DATA_BLOCK DB 3
AUTHOR : sra
FAMILY : AZO
VERSION : 0.0
  STRUCT
   OB1_Info : STRUCT
    OB1_DATE_TIME : DATE_AND_TIME ;	//Date and time OB1 started
    OB1_PREV_CYCLE : INT ;	//Cycle time of previous OB1 scan (milliseconds)
    OB1_MIN_CYCLE : INT ;	//Minimum cycle time of OB1 (milliseconds)
    OB1_MAX_CYCLE : INT ;	//Maximum cycle time of OB1 (milliseconds)
    reserve : ARRAY  [0 .. 14 ] OF BYTE ;
   END_STRUCT ;
   Fehler_OB_Info : STRUCT
    Zeitfehler_OB80 : BOOL ;	//Zeitfehler OB 80
    Stromversorgung_OB81 : BOOL ;	//Stromversorgungsfehler OB 81
    Diagnose_Alarm_OB82 : BOOL ;	//Diagnose-Alarm OB82
    Ziehen_Stecken_OB83 : BOOL ;	//Ziehen/Stecken-Alarm OB83
    CPU_Hardware_OB84 : BOOL ;	//CPU-Hardwarefehler OB84
    Programmablauf_OB85 : BOOL ;	//Programmablauffehler OB85
    Baugr_tr_ausfall_OB86 : BOOL ;	//Baugruppenträgerausfall OB86
    Kommunikation_OB87 : BOOL ;	//Kommunikationsfehler OB87
    Programmierfehler_OB121 : BOOL ;	//Programmierfehler OB121
    Periphzugriff_OB122 : BOOL ;	//Peripheriezugriffsfehler OB 122
    Bearbeitungsabbruch_OB88 : BOOL ;	//Bearbeitungsabbruch eines Bausteins OB88
    Battery_fault : BOOL ;	//Battery fault with SFC51
    reserve_word : WORD ;
    OB_80_Fault_ID : BYTE ;	//Fehlercode OB 80
    OB_81_Fault_ID : BYTE ;	//Fehlercode OB 81
    OB_82_Fault_ID : BYTE ;	//Fehlercode OB 82
    OB_83_Fault_ID : BYTE ;	//Fehlercode OB 83
    OB_84_Fault_ID : BYTE ;	//Fehlercode OB 84
    OB_85_Fault_ID : BYTE ;	//Fehlercode OB 85
    OB_86_Fault_ID : BYTE ;	//Fehlercode OB 86
    OB_87_Fault_ID : BYTE ;	//Fehlercode OB 87
    OB_121_Fault_ID : BYTE ;	//Fehlercode OB 121
    OB_122_Fault_ID : BYTE ;	//Fehlercode OB 122
    OB_88_Fault_ID : BYTE ;	//Fehlercode OB 122
    reserve : ARRAY  [16 .. 29 ] OF BYTE ;
   END_STRUCT ;
   RDSYSST : STRUCT
    BUSY : BOOL ;
    RETVAL : INT ;
    SLZ_HEADER : STRUCT
     LENTHDR : WORD ;
     N_DR : WORD ;
    END_STRUCT ;
    DR : STRUCT
     Data_1 : BYTE ;
     Data_2 : BYTE ;
     Data_3 : BYTE ;
     Data_4 : BYTE ;
     Data_5 : BYTE ;
     Data_6 : BYTE ;
     Data_7 : BYTE ;
     Data_8 : BYTE ;
     Data_9 : BYTE ;
     Data_10 : BYTE ;
     Data_11 : BYTE ;
     Data_12 : BYTE ;
     Data_13 : BYTE ;
     Data_14 : BYTE ;
     Data_15 : BYTE ;
     Data_16 : BYTE ;
     Data_17 : BYTE ;
     Data_18 : BYTE ;
     Data_19 : BYTE ;
     Data_20 : BYTE ;
    END_STRUCT ;
   END_STRUCT ;
  END_STRUCT ;	
BEGIN
END_DATA_BLOCK

DATA_BLOCK DB 4
VERSION : 0.1
  STRUCT
   Motordaten1 : STRUCT 	//Anzahl der Motordaten abhängig von der Anzahl der verschied. benutzten Motoren
    Nennleistungsfaktor : REAL  := 8.000000e-001;	//Motornennleistungsfaktor cos phi
    Nennfrequenz : REAL  := 5.100000e+001;	//Motornennfrequenz in Einheit Hz
    Nenndrehzahl : REAL  := 1.400000e+003;	//Motornenndrehzal in U/min
    Nennstrom : REAL  := 6.100000e+000;	//Motornennstrom in A
    Nennspannung : REAL  := 2.310000e+002;	//Motornennspannung in V
    Nennleistung : REAL  := 1.400000e+000;	//Motornennleistung kW
    reserve : ARRAY  [24 .. 29 ] OF //Reserve für weitere Motordaten
    BYTE ;
   END_STRUCT ;
   Motordaten2 : STRUCT
    Nennleistungsfaktor : REAL  := 7.000000e-001;
    Nennfrequenz : REAL  := 1.000000e+002;
    Nenndrehzahl : REAL  := 2.000000e+002;
    Nennstrom : REAL  := 2.000000e+000;
    Nennspannung : REAL  := 3.800000e+002;
    Nennleistung : REAL  := 1.000000e+003;
    reserve : ARRAY  [24 .. 29 ] OF BYTE ;
   END_STRUCT ;
   Motordaten3 : STRUCT
    Nennleistungsfaktor : REAL  := 7.000000e-001;
    Nennfrequenz : REAL  := 1.000000e+002;
    Nenndrehzahl : REAL  := 2.000000e+002;
    Nennstrom : REAL  := 5.000000e+000;
    Nennspannung : REAL  := 3.800000e+002;
    Nennleistung : REAL  := 1.000000e+003;
    reserve : ARRAY  [24 .. 29 ] OF BYTE ;
   END_STRUCT ;
   Motordaten4 : STRUCT
    Nennleistungsfaktor : REAL  := 7.000000e-001;
    Nennfrequenz : REAL  := 1.000000e+002;
    Nenndrehzahl : REAL  := 2.000000e+002;
    Nennstrom : REAL  := 5.000000e+000;
    Nennspannung : REAL  := 3.800000e+002;
    Nennleistung : REAL  := 1.000000e+003;
    reserve : ARRAY  [24 .. 29 ] OF BYTE ;
   END_STRUCT ;
   Motordaten5 : STRUCT
    Nennleistungsfaktor : REAL  := 7.000000e-001;
    Nennfrequenz : REAL  := 1.000000e+002;
    Nenndrehzahl : REAL  := 2.000000e+002;
    Nennstrom : REAL  := 5.000000e+000;
    Nennspannung : REAL  := 3.800000e+002;
    Nennleistung : REAL  := 1.000000e+003;
    reserve : ARRAY  [24 .. 29 ] OF BYTE ;
   END_STRUCT ;
   Motordaten6 : STRUCT
    Nennleistungsfaktor : REAL  := 7.000000e-001;
    Nennfrequenz : REAL  := 1.000000e+002;
    Nenndrehzahl : REAL  := 2.000000e+002;
    Nennstrom : REAL  := 5.000000e+000;
    Nennspannung : REAL  := 3.800000e+002;
    Nennleistung : REAL  := 1.000000e+003;
    reserve : ARRAY  [24 .. 29 ] OF BYTE ;
   END_STRUCT ;
   Motordaten7 : STRUCT
    Nennleistungsfaktor : REAL  := 7.000000e-001;
    Nennfrequenz : REAL  := 1.000000e+002;
    Nenndrehzahl : REAL  := 2.000000e+002;
    Nennstrom : REAL  := 5.000000e+000;
    Nennspannung : REAL  := 3.800000e+002;
    Nennleistung : REAL  := 1.000000e+003;
    reserve : ARRAY  [24 .. 29 ] OF BYTE ;
   END_STRUCT ;
   Motordaten8 : STRUCT
    Nennleistungsfaktor : REAL  := 7.000000e-001;
    Nennfrequenz : REAL  := 1.000000e+002;
    Nenndrehzahl : REAL  := 2.000000e+002;
    Nennstrom : REAL  := 5.000000e+000;
    Nennspannung : REAL  := 3.800000e+002;
    Nennleistung : REAL  := 1.000000e+003;
    reserve : ARRAY  [24 .. 29 ] OF BYTE ;
   END_STRUCT ;
   Motordaten9 : STRUCT
    Nennleistungsfaktor : REAL  := 7.000000e-001;
    Nennfrequenz : REAL  := 1.000000e+002;
    Nenndrehzahl : REAL  := 2.000000e+002;
    Nennstrom : REAL  := 5.000000e+000;
    Nennspannung : REAL  := 3.800000e+002;
    Nennleistung : REAL  := 1.000000e+003;
    reserve : ARRAY  [24 .. 29 ] OF BYTE ;
   END_STRUCT ;
   Motordaten10 : STRUCT
    Nennleistungsfaktor : REAL  := 7.000000e-001;
    Nennfrequenz : REAL  := 1.000000e+002;
    Nenndrehzahl : REAL  := 2.000000e+002;
    Nennstrom : REAL  := 5.000000e+000;
    Nennspannung : REAL  := 3.800000e+002;
    Nennleistung : REAL  := 1.000000e+003;
    reserve : ARRAY  [24 .. 29 ] OF BYTE ;
   END_STRUCT ;
  END_STRUCT ;	
BEGIN
   Motordaten1.Nennleistungsfaktor := 8.000000e-01;
   Motordaten1.Nennfrequenz := 5.100000e+01;
   Motordaten1.Nenndrehzahl := 1.400000e+03;
   Motordaten1.Nennstrom := 6.100000e+00;
   Motordaten1.Nennspannung := 2.310000e+02;
   Motordaten1.Nennleistung := 1.400000e+00;
   Motordaten2.Nennleistungsfaktor := 7.000000e-01;
   Motordaten2.Nennfrequenz := 1.000000e+02;
   Motordaten2.Nenndrehzahl := 2.000000e+02;
   Motordaten2.Nennstrom := 5.000000e+00;
   Motordaten2.Nennspannung := 3.800000e+02;
   Motordaten2.Nennleistung := 1.000000e+03;
   Motordaten3.Nennleistungsfaktor := 7.000000e-01;
   Motordaten3.Nennfrequenz := 1.000000e+02;
   Motordaten3.Nenndrehzahl := 2.000000e+02;
   Motordaten3.Nennstrom := 5.000000e+00;
   Motordaten3.Nennspannung := 3.800000e+02;
   Motordaten3.Nennleistung := 1.000000e+03;
   Motordaten4.Nennleistungsfaktor := 7.000000e-01;
   Motordaten4.Nennfrequenz := 1.000000e+02;
   Motordaten4.Nenndrehzahl := 2.000000e+02;
   Motordaten4.Nennstrom := 5.000000e+00;
   Motordaten4.Nennspannung := 3.800000e+02;
   Motordaten4.Nennleistung := 1.000000e+03;
   Motordaten5.Nennleistungsfaktor := 7.000000e-01;
   Motordaten5.Nennfrequenz := 1.000000e+02;
   Motordaten5.Nenndrehzahl := 2.000000e+02;
   Motordaten5.Nennstrom := 5.000000e+00;
   Motordaten5.Nennspannung := 3.800000e+02;
   Motordaten5.Nennleistung := 1.000000e+03;
   Motordaten6.Nennleistungsfaktor := 7.000000e-01;
   Motordaten6.Nennfrequenz := 1.000000e+02;
   Motordaten6.Nenndrehzahl := 2.000000e+02;
   Motordaten6.Nennstrom := 5.000000e+00;
   Motordaten6.Nennspannung := 3.800000e+02;
   Motordaten6.Nennleistung := 1.000000e+03;
   Motordaten7.Nennleistungsfaktor := 7.000000e-01;
   Motordaten7.Nennfrequenz := 1.000000e+02;
   Motordaten7.Nenndrehzahl := 2.000000e+02;
   Motordaten7.Nennstrom := 5.000000e+00;
   Motordaten7.Nennspannung := 3.800000e+02;
   Motordaten7.Nennleistung := 1.000000e+03;
   Motordaten8.Nennleistungsfaktor := 7.000000e-01;
   Motordaten8.Nennfrequenz := 1.000000e+02;
   Motordaten8.Nenndrehzahl := 2.000000e+02;
   Motordaten8.Nennstrom := 5.000000e+00;
   Motordaten8.Nennspannung := 3.800000e+02;
   Motordaten8.Nennleistung := 1.000000e+03;
   Motordaten9.Nennleistungsfaktor := 7.000000e-01;
   Motordaten9.Nennfrequenz := 1.000000e+02;
   Motordaten9.Nenndrehzahl := 2.000000e+02;
   Motordaten9.Nennstrom := 5.000000e+00;
   Motordaten9.Nennspannung := 3.800000e+02;
   Motordaten9.Nennleistung := 1.000000e+03;
   Motordaten10.Nennleistungsfaktor := 7.000000e-01;
   Motordaten10.Nennfrequenz := 1.000000e+02;
   Motordaten10.Nenndrehzahl := 2.000000e+02;
   Motordaten10.Nennstrom := 5.000000e+00;
   Motordaten10.Nennspannung := 3.800000e+02;
   Motordaten10.Nennleistung := 1.000000e+03;
END_DATA_BLOCK

DATA_BLOCK DB 30
AUTHOR : sra
FAMILY : hsh
VERSION : 0.0
FB 30
BEGIN
END_DATA_BLOCK

DATA_BLOCK DB 32
AUTHOR : sra
FAMILY : SCADA
VERSION : 0.0
FB 32
BEGIN
END_DATA_BLOCK

DATA_BLOCK DB 33
AUTHOR : sra
FAMILY : SCADA
VERSION : 0.0
FB 33
BEGIN
END_DATA_BLOCK

DATA_BLOCK DB 34
AUTHOR : sra
FAMILY : AZO
VERSION : 0.0
FB 34
BEGIN
END_DATA_BLOCK

DATA_BLOCK DB 35
VERSION : 0.1
  STRUCT
   Quittierung : ARRAY  [0 .. 1023, 0 .. 7 ] OF BOOL  := FALSE;
   Quittierung_Spiegelungen : ARRAY  [0 .. 1023, 0 .. 7 ] OF BOOL  := FALSE;
  END_STRUCT ;	
BEGIN
END_DATA_BLOCK

DATA_BLOCK DB 92
VERSION : 0.0
FB 92
BEGIN
END_DATA_BLOCK

DATA_BLOCK DB 1000
AUTHOR : ilia
VERSION : 0.0
FB 1000
BEGIN
END_DATA_BLOCK

DATA_BLOCK DB 1001
AUTHOR : ilia
VERSION : 0.1
FB 1001
BEGIN
END_DATA_BLOCK

DATA_BLOCK DB 1011
AUTHOR : ilia
VERSION : 0.1
FB 1011
BEGIN
END_DATA_BLOCK

DATA_BLOCK DB 1051
AUTHOR : ilia
VERSION : 0.1
FB 1051
BEGIN
END_DATA_BLOCK

DATA_BLOCK DB 1111
VERSION : 0.1
  STRUCT
   RECIPE1 : STRUCT 	//Recipe
    RecipeName : STRING  [18 ] := 'RECIPE1';	//Recipe Name
    SpeedRinne : INT  := 30;	//Speed of Rinne
    SpeedRotaryFeeder : INT  := 30;	//Speed of RF
    SpeedVacuumPump : INT  := 35;	//Speed of VP1
    NumberOfPumps : INT  := 1;
    reserve1 : INT ;
    reserve2 : INT ;
    reserve3 : ARRAY  [1 .. 8 ] OF BYTE  := B#16#0;
   END_STRUCT ;
   RECIPE2 : STRUCT 	//Recipe
    RecipeName : STRING  [18 ] := 'RECIPE2';	//Recipe Name
    SpeedRinne : INT  := 30;	//Speed of Rinne
    SpeedRotaryFeeder : INT  := 30;	//Speed of RF
    SpeedVacuumPump : INT  := 35;	//Speed of VP1
    NumberOfPumps : INT  := 1;
    reserve1 : INT ;
    reserve2 : INT ;
    reserve3 : ARRAY  [1 .. 8 ] OF BYTE  := B#16#0;
   END_STRUCT ;
   RECIPE3 : STRUCT 	//Recipe
    RecipeName : STRING  [18 ] := 'RECIPE3';	//Recipe Name
    SpeedRinne : INT  := 30;	//Speed of Rinne
    SpeedRotaryFeeder : INT  := 30;	//Speed of RF
    SpeedVacuumPump : INT  := 35;	//Speed of VP1
    NumberOfPumps : INT  := 1;
    reserve1 : INT ;
    reserve2 : INT ;
    reserve3 : ARRAY  [1 .. 8 ] OF BYTE  := B#16#0;
   END_STRUCT ;
   RECIPE4 : STRUCT 	//Recipe
    RecipeName : STRING  [18 ] := 'RECIPE4';	//Recipe Name
    SpeedRinne : INT  := 30;	//Speed of Rinne
    SpeedRotaryFeeder : INT  := 30;	//Speed of RF
    SpeedVacuumPump : INT  := 35;	//Speed of VP1
    NumberOfPumps : INT  := 1;
    reserve1 : INT ;
    reserve2 : INT ;
    reserve3 : ARRAY  [1 .. 8 ] OF BYTE  := B#16#0;
   END_STRUCT ;
   RECIPE5 : STRUCT 	//Recipe
    RecipeName : STRING  [18 ] := 'RECIPE5';	//Recipe Name
    SpeedRinne : INT  := 30;	//Speed of Rinne
    SpeedRotaryFeeder : INT  := 30;	//Speed of RF
    SpeedVacuumPump : INT  := 35;	//Speed of VP1
    NumberOfPumps : INT  := 1;
    reserve1 : INT ;
    reserve2 : INT ;
    reserve3 : ARRAY  [1 .. 8 ] OF BYTE  := B#16#0;
   END_STRUCT ;
   RECIPE6 : STRUCT 	//Recipe
    RecipeName : STRING  [18 ] := 'RECIPE6';	//Recipe Name
    SpeedRinne : INT  := 30;	//Speed of Rinne
    SpeedRotaryFeeder : INT  := 30;	//Speed of RF
    SpeedVacuumPump : INT  := 35;	//Speed of VP1
    NumberOfPumps : INT  := 1;
    reserve1 : INT ;
    reserve2 : INT ;
    reserve3 : ARRAY  [1 .. 8 ] OF BYTE  := B#16#0;
   END_STRUCT ;
   RECIPE7 : STRUCT 	//Recipe
    RecipeName : STRING  [18 ] := 'RECIPE7';	//Recipe Name
    SpeedRinne : INT  := 30;	//Speed of Rinne
    SpeedRotaryFeeder : INT  := 30;	//Speed of RF
    SpeedVacuumPump : INT  := 35;	//Speed of VP1
    NumberOfPumps : INT  := 1;
    reserve1 : INT ;
    reserve2 : INT ;
    reserve3 : ARRAY  [1 .. 8 ] OF BYTE  := B#16#0;
   END_STRUCT ;
   RECIPE8 : STRUCT 	//Recipe
    RecipeName : STRING  [18 ] := 'RECIPE8';	//Recipe Name
    SpeedRinne : INT  := 30;	//Speed of Rinne
    SpeedRotaryFeeder : INT  := 30;	//Speed of RF
    SpeedVacuumPump : INT  := 35;	//Speed of VP1
    NumberOfPumps : INT  := 1;
    reserve1 : INT ;
    reserve2 : INT ;
    reserve3 : ARRAY  [1 .. 8 ] OF BYTE  := B#16#0;
   END_STRUCT ;
   RECIPE9 : STRUCT 	//Recipe
    RecipeName1 : STRING  [18 ] := 'RECIPE9';	//Recipe Name
    SpeedRinne : INT  := 30;	//Speed of Rinne
    SpeedRotaryFeeder : INT  := 30;	//Speed of RF
    SpeedVacuumPump : INT  := 35;	//Speed of VP1
    NumberOfPumps : INT  := 1;
    reserve1 : INT ;
    reserve2 : INT ;
    reserve3 : ARRAY  [1 .. 8 ] OF BYTE  := B#16#0;
   END_STRUCT ;
   RECIPE10 : STRUCT 	//Recipe
    RecipeName : STRING  [18 ] := 'RECIPE10';	//Recipe Name
    SpeedRinne : INT  := 30;	//Speed of Rinne
    SpeedRotaryFeeder : INT  := 30;	//Speed of RF
    SpeedVacuumPump : INT  := 35;	//Speed of VP1
    NumberOfPumps : INT  := 1;
    reserve1 : INT ;
    reserve2 : INT ;
    reserve3 : ARRAY  [1 .. 8 ] OF BYTE  := B#16#0;
   END_STRUCT ;
  END_STRUCT ;	
BEGIN
   RECIPE1.RecipeName := 'RECIPE1';
   RECIPE1.SpeedRinne := 30;
   RECIPE1.SpeedRotaryFeeder := 30;
   RECIPE1.SpeedVacuumPump := 35;
   RECIPE1.NumberOfPumps := 1;
   RECIPE2.RecipeName := 'RECIPE2';
   RECIPE2.SpeedRinne := 30;
   RECIPE2.SpeedRotaryFeeder := 30;
   RECIPE2.SpeedVacuumPump := 35;
   RECIPE2.NumberOfPumps := 1;
   RECIPE3.RecipeName := 'RECIPE3';
   RECIPE3.SpeedRinne := 30;
   RECIPE3.SpeedRotaryFeeder := 30;
   RECIPE3.SpeedVacuumPump := 35;
   RECIPE3.NumberOfPumps := 1;
   RECIPE4.RecipeName := 'RECIPE4';
   RECIPE4.SpeedRinne := 30;
   RECIPE4.SpeedRotaryFeeder := 30;
   RECIPE4.SpeedVacuumPump := 35;
   RECIPE4.NumberOfPumps := 1;
   RECIPE5.RecipeName := 'RECIPE5';
   RECIPE5.SpeedRinne := 30;
   RECIPE5.SpeedRotaryFeeder := 30;
   RECIPE5.SpeedVacuumPump := 35;
   RECIPE5.NumberOfPumps := 1;
   RECIPE6.RecipeName := 'RECIPE6';
   RECIPE6.SpeedRinne := 30;
   RECIPE6.SpeedRotaryFeeder := 30;
   RECIPE6.SpeedVacuumPump := 35;
   RECIPE6.NumberOfPumps := 1;
   RECIPE7.RecipeName := 'RECIPE7';
   RECIPE7.SpeedRinne := 30;
   RECIPE7.SpeedRotaryFeeder := 30;
   RECIPE7.SpeedVacuumPump := 35;
   RECIPE7.NumberOfPumps := 1;
   RECIPE8.RecipeName := 'RECIPE8';
   RECIPE8.SpeedRinne := 30;
   RECIPE8.SpeedRotaryFeeder := 30;
   RECIPE8.SpeedVacuumPump := 35;
   RECIPE8.NumberOfPumps := 1;
   RECIPE9.RecipeName1 := 'RECIPE9';
   RECIPE9.SpeedRinne := 30;
   RECIPE9.SpeedRotaryFeeder := 30;
   RECIPE9.SpeedVacuumPump := 35;
   RECIPE9.NumberOfPumps := 1;
   RECIPE10.RecipeName := 'RECIPE10';
   RECIPE10.SpeedRinne := 30;
   RECIPE10.SpeedRotaryFeeder := 30;
   RECIPE10.SpeedVacuumPump := 35;
   RECIPE10.NumberOfPumps := 1;
END_DATA_BLOCK

DATA_BLOCK DB 2222
VERSION : 0.1
  STRUCT
   Recipe : STRUCT 	//Temporary placeholder variable
    Speed_1 : INT  := 1;
    Speed_2 : INT  := 2;
    Number : INT ;
   END_STRUCT ;
  END_STRUCT ;	
BEGIN
   Recipe.Speed_1 := 1;
   Recipe.Speed_2 := 2;
END_DATA_BLOCK

DATA_BLOCK DB 4900
AUTHOR : ilia
VERSION : 0.0
FB 4900
BEGIN
END_DATA_BLOCK

DATA_BLOCK DB 10001
VERSION : 0.0
FB 4901
BEGIN
END_DATA_BLOCK

DATA_BLOCK DB 10002
VERSION : 0.0
FB 4901
BEGIN
END_DATA_BLOCK

ORGANIZATION_BLOCK OB 1
TITLE = zyklischer Programmablauf
//Erstellung:
//Datum        Bearbeiter                                                 Version
//--------------------------------------------------------------------------------
//01.08.18     Ilia Bedniakov                                             01.00.00
//
//Änderungen:
//Nr. Datum    Bearb Beschreibung                                   Marke Version
//--------------------------------------------------------------------------------
//01  
//
VERSION : 0.1
VAR_TEMP
  OB1_EV_CLASS : BYTE ;	//Bits 0-3 = 1 (Coming event), Bits 4-7 = 1 (Event class 1)
  OB1_SCAN_1 : BYTE ;	//1 (Cold restart scan 1 of OB 1), 3 (Scan 2-n of OB 1)
  OB1_PRIORITY : BYTE ;	//1 (Priority of 1 is lowest)
  OB1_OB_NUMBR : BYTE ;	//1 (Organization block 1, OB1)
  OB1_RESERVED_1 : BYTE ;	//Reserved for system
  OB1_RESERVED_2 : BYTE ;	//Reserved for system
  OB1_PREV_CYCLE : INT ;	//Cycle time of previous OB1 scan (milliseconds)
  OB1_MIN_CYCLE : INT ;	//Minimum cycle time of OB1 (milliseconds)
  OB1_MAX_CYCLE : INT ;	//Maximum cycle time of OB1 (milliseconds)
  OB1_DATE_TIME : DATE_AND_TIME ;	//Date and time OB1 started
  DUMMY_INT : INT ;
  dummybool : BOOL ;
END_VAR
BEGIN
NETWORK
TITLE = Simulation
//      CLR   
      SET;
      =     M 0.5;
      A     M 0.5;
      JCN   NS;	// No simulation
      CALL  FB 2 , DB 2;
NS:   NOP   0;
NETWORK
TITLE = Datum, Uhrzeit und Zykluszeiten in DB3 kopieren
      CALL  SFC 20 (
           SRCBLK                   := #OB1_DATE_TIME,
           RET_VAL                  := #DUMMY_INT,
           DSTBLK                   := P#DB3.DBX 0.0 BYTE 8);
      L     #OB1_PREV_CYCLE;
      T     DB3.DBW 8;
      L     #OB1_MIN_CYCLE;
      T     DB3.DBW 10;
      L     #OB1_MAX_CYCLE;
      T     DB3.DBW 12;
NETWORK
TITLE = Standardsignale
      CALL  FC 13 (
           in_E_Sicherung_OK        := I 5.7,
           in_Basistakt_Timer       := M 4.1,
           in_Zeit_Basistakt_100ms  := 2,
           o_Lampe_Stoer_Sicherung  := #dummybool,
           o_Stoerung_Sicherung     := #dummybool);
NETWORK
TITLE = Daten von/an HMI
      CALL  FB 30 , DB 30;
      CALL  FB 32 , DB 32;
      CALL  FB 33 , DB 33;
NETWORK
TITLE = Stoerungen Auswertung
      CALL  FB 34 , DB 34;
NETWORK
TITLE = Anwenderprogramm
      CALL  FB 1000 , DB 1000;
NETWORK
TITLE = Neustart oder Wiederanlauf SPS rücksetzen
//letztes Netzwerk
      SET;
      R     M 1.3;
      R     M 1.4;
END_ORGANIZATION_BLOCK

ORGANIZATION_BLOCK OB 80
TITLE = Zeitfehler
//Erstellung:
//Datum        Bearbeiter                                                 Version
//--------------------------------------------------------------------------------
//03.06.98     Rainer Schaffert (sra)                                     01.00.00
//
//Änderungen:
//Nr. Datum    Bearb Beschreibung                                   Marke Version
//--------------------------------------------------------------------------------
//01  
//
//________________________________________________________________________________
//OB wird bei Zeitfehler bearbeitet
//
AUTHOR : sra
FAMILY : error_OB
NAME : time_err
VERSION : 0.1
VAR_TEMP
  OB80_EV_CLASS : BYTE ;	//16#35, Event class 3, Entering event state, Internal fault event
  OB80_FLT_ID : BYTE ;	//16#XX, Fault identifcation code
  OB80_PRIORITY : BYTE ;	//26 (Priority of 1 is lowest)
  OB80_OB_NUMBR : BYTE ;	//80 (Organization block 80, OB80)
  OB80_RESERVED_1 : BYTE ;	//Reserved for system
  OB80_RESERVED_2 : BYTE ;	//Reserved for system
  OB80_ERROR_INFO : WORD ;	//Error information on event
  OB80_ERR_EV_CLASS : BYTE ;	//Class of event causing error
  OB80_ERR_EV_NUM : BYTE ;	//Number of event causing error
  OB80_OB_PRIORITY : BYTE ;	//Priority of OB causing error
  OB80_OB_NUM : BYTE ;	//Number of OB causing error
  OB80_DATE_TIME : DATE_AND_TIME ;	//Date and time OB80 started
END_VAR
BEGIN
NETWORK
TITLE = Fehlermeldung erzeugen
//Fehlermeldung erzeugen
//
//Fehlercode B#16#01 : Zykluszeit überschritten
//                     OB80_ERROR_INFO: Laufzeit des letzten Zyklus
//           
//           B#16#02 : Der angeforderte OB ist noch in Bearbeitung
//
//           B#16#07 : Überlauf des OB-Anforderungspuffers für die aktuelle 
//                     Prioritätsklasse
//
//           B#16#05 : abgelaufener Urzeitalarm durch Urzeitsprung
//
//           B#16#06 : abgelaufener Urzeitalarm bei Wiedereintritt 
//
      L     #OB80_FLT_ID;
      L     B#16#0;
      <>I;
      =     DB3.DBX 30.0;
      L     #OB80_FLT_ID;
      T     DB3.DBB 34;
END_ORGANIZATION_BLOCK

ORGANIZATION_BLOCK OB 82
TITLE = Diagnose-Alarm
//Erstellung:
//Datum        Bearbeiter                                                 Version
//--------------------------------------------------------------------------------
//03.06.98     Rainer Schaffert (sra)                                     01.00.00
//
//Änderungen:
//Nr. Datum    Bearb Beschreibung                                   Marke Version
//--------------------------------------------------------------------------------
//01  
//
//________________________________________________________________________________
//OB wird bei Diagnose-Alarm bearbeitet
//
AUTHOR : sra
FAMILY : error_OB
NAME : diagn_OB
VERSION : 0.1
VAR_TEMP
  OB82_EV_CLASS : BYTE ;	//16#39, Event class 3, Entering event state, Internal fault event
  OB82_FLT_ID : BYTE ;	//16#XX, Fault identifcation code
  OB82_PRIORITY : BYTE ;	//26/28 (Priority of 1 is lowest)
  OB82_OB_NUMBR : BYTE ;	//82 (Organization block 82, OB82)
  OB82_RESERVED_1 : BYTE ;	//Reserved for system
  OB82_IO_FLAG : BYTE ;	//Input (01010100), Output (01010101)
  OB82_MDL_ADDR : INT ;	//Base address of module with fault
  OB82_MDL_DEFECT : BOOL ;	//Module defective
  OB82_INT_FAULT : BOOL ;	//Internal fault
  OB82_EXT_FAULT : BOOL ;	//External fault
  OB82_PNT_INFO : BOOL ;	//Point information
  OB82_EXT_VOLTAGE : BOOL ;	//External voltage low
  OB82_FLD_CONNCTR : BOOL ;	//Field wiring connector missing
  OB82_NO_CONFIG : BOOL ;	//Module has no configuration data
  OB82_CONFIG_ERR : BOOL ;	//Module has configuration error
  OB82_MDL_TYPE : BYTE ;	//Type of module
  OB82_SUB_NDL_ERR : BOOL ;	//Sub-Module is missing or has error
  OB82_COMM_FAULT : BOOL ;	//Communication fault
  OB82_MDL_STOP : BOOL ;	//Module is stopped
  OB82_WTCH_DOG_FLT : BOOL ;	//Watch dog timer stopped module
  OB82_INT_PS_FLT : BOOL ;	//Internal power supply fault
  OB82_PRIM_BATT_FLT : BOOL ;	//Primary battery is in fault
  OB82_BCKUP_BATT_FLT : BOOL ;	//Backup battery is in fault
  OB82_RESERVED_2 : BOOL ;	//Reserved for system
  OB82_RACK_FLT : BOOL ;	//Rack fault, only for bus interface module
  OB82_PROC_FLT : BOOL ;	//Processor fault
  OB82_EPROM_FLT : BOOL ;	//EPROM fault
  OB82_RAM_FLT : BOOL ;	//RAM fault
  OB82_ADU_FLT : BOOL ;	//ADU fault
  OB82_FUSE_FLT : BOOL ;	//Fuse fault
  OB82_HW_INTR_FLT : BOOL ;	//Hardware interupt input in fault
  OB82_RESERVED_3 : BOOL ;	//Reserved for system
  OB82_DATE_TIME : DATE_AND_TIME ;	//Date and time OB82 started
END_VAR
BEGIN
NETWORK
TITLE = Fehlermeldung erzeugen
//Fehlermeldung erzeugen
//
//Fehlercode B#16#42 : 
//
      A(;
      L     #OB82_EV_CLASS;
      L     B#16#39;	// kommendes Ereignis
      ==I;
      );
      A(;
      L     #OB82_FLT_ID;
      L     B#16#0;
      <>I;
      );
      =     DB3.DBX 30.2;
      L     #OB82_FLT_ID;
      T     DB3.DBB 36;
END_ORGANIZATION_BLOCK

ORGANIZATION_BLOCK OB 83
TITLE = Ziehen/Stecken-Alarm
//Erstellung:
//Datum        Bearbeiter                                                 Version
//--------------------------------------------------------------------------------
//03.06.98     Rainer Schaffert (sra)                                     01.00.00
//
//Änderungen:
//Nr. Datum    Bearb Beschreibung                                   Marke Version
//--------------------------------------------------------------------------------
//01  
//
//________________________________________________________________________________
//OB wird bei Ziehen/Stecken-Alarm bearbeitet
//
AUTHOR : sra
FAMILY : AZO
VERSION : 0.0
VAR_TEMP
  OB83_EV_CLASS : BYTE ;	//16#38/39, Event class 3, module inserted/removed (8/9)
  OB83_FLT_ID : BYTE ;	//16#XX, Fault identifcation code
  OB83_PRIORITY : BYTE ;	//26/28 (Priority of 1 is lowest)
  OB83_OB_NUMBR : BYTE ;	//83 (Organization block 83, OB83)
  OB83_RESERVED_1 : BYTE ;	//Reserved for system
  OB83_MDL_ID : BYTE ;	//Input module (01010100), Output module (01010101)
  OB83_MDL_ADDR : WORD ;	//Base address of module with point fault
  OB83_RACK_NUM : WORD ;	//Number of rack that has module with point fault
  OB83_MDL_TYPE : WORD ;	//Module type with point fault
  OB83_DATE_TIME : DATE_AND_TIME ;	//Date and time OB83 started
END_VAR
BEGIN
NETWORK
TITLE = Fehlermeldung erzeugen
//Fehlermeldung erzeugen
//
//Fehlercode B#16#61 : Baugruppe gezogen bzw. nicht ansprechbar (bei 
//                     Ereignisklasse B#16#39)
//                     Baugruppe gesteckt, Baugruppentyp ok (bei
//                     Ereignisklasse B#16#38)
//           
//           B#16#63 : Baugruppe gesteckt, jedoch falscher Baugruppentyp
//
//           B#16#64 : Baugruppe gesteckt, jedoch gestört(Typkennung nicht lesbar)
//
      A(;
      L     #OB83_EV_CLASS;
      L     B#16#39;	// kommendes Ereignis
      ==I;
      );
      A(;
      L     #OB83_FLT_ID;
      L     B#16#0;
      <>I;
      );
      =     DB3.DBX 30.3;
      L     #OB83_FLT_ID;
      T     DB3.DBB 37;
END_ORGANIZATION_BLOCK

ORGANIZATION_BLOCK OB 85
TITLE = Programmablauffehler
//Erstellung:
//Datum        Bearbeiter                                                 Version
//--------------------------------------------------------------------------------
//03.06.98     Rainer Schaffert (sra)                                     01.00.00
//
//Änderungen:
//Nr. Datum    Bearb Beschreibung                                   Marke Version
//--------------------------------------------------------------------------------
//01  
//
//________________________________________________________________________________
//OB wird bei Programmablauffehler bearbeitet
//
//
AUTHOR : sra
FAMILY : AZO
VERSION : 0.0
VAR_TEMP
  OB85_EV_CLASS : BYTE ;	//16#35 Event class 3
  OB85_FLT_ID : BYTE ;	//16#XX, Fault identification code
  OB85_PRIORITY : BYTE ;	//26 (Priority of 1 is lowest)
  OB85_OB_NUMBR : BYTE ;	//85 (Organization block 85, OB85)
  OB85_RESERVED_1 : BYTE ;	//Reserved for system
  OB85_RESERVED_2 : BYTE ;	//Reserved for system
  OB85_RESERVED_3 : INT ;	//Reserved for system
  OB85_ERR_EV_CLASS : BYTE ;	//Class of event causing error
  OB85_ERR_EV_NUM : BYTE ;	//Number of event causing error
  OB85_OB_PRIOR : BYTE ;	//Priority of OB causing error
  OB85_OB_NUM : BYTE ;	//Number of OB causing error
  OB85_DATE_TIME : DATE_AND_TIME ;	//Date and time OB85 started
END_VAR
BEGIN
NETWORK
TITLE = Fehlermeldung erzeugen
//Fehlermeldung erzeugen
//
//Fehlercode B#16#A1 : Das Programm oder das Betriebssystem erzeugt ein 
//                     Startereignis für einen OB, der nicht in die CPU geladen 
//                     ist.
//
//           B#16#A2 : Das Programm oder das Betriebssystem erzeugt ein 
//                     Startereignis für einen OB, der nicht in die CPU geladen 
//                     ist.
//
//           B#16#A3 : Fehler beim Zugriff des Betriebssystems auf einen Baustein
//
//           B#16#B1 : Peripheriezugriffsfehler beim Aktualisieren des 
//                     Gesamtprozessabbildes der Eingänge
//
//           B#16#B1 : Peripheriezugriffsfehler beim Aktualisieren des            
//                     Gesamtprozessabbildes der Ausgänge
//
      L     #OB85_FLT_ID;
      L     B#16#0;
      <>I;
      =     DB3.DBX 30.5;
      L     #OB85_FLT_ID;
      T     DB3.DBB 39;
END_ORGANIZATION_BLOCK

ORGANIZATION_BLOCK OB 86
TITLE = Baugruppenträgerausfall
//Erstellung:
//Datum        Bearbeiter                                                 Version
//--------------------------------------------------------------------------------
//03.06.98     Rainer Schaffert (sra)                                     01.00.00
//
//Änderungen:
//Nr. Datum    Bearb Beschreibung                                   Marke Version
//--------------------------------------------------------------------------------
//01  
//
//________________________________________________________________________________
//OB wird bei Baugruppenträgerausfall bearbeitet
//
AUTHOR : sra
FAMILY : AZO
VERSION : 0.0
VAR_TEMP
  OB86_EV_CLASS : BYTE ;	//16#38/39 Event class 3
  OB86_FLT_ID : BYTE ;	//16#C1/C4/C5, Fault identification code
  OB86_PRIORITY : BYTE ;	//26/28 (Priority of 1 is lowest)
  OB86_OB_NUMBR : BYTE ;	//86 (Organization block 86, OB86)
  OB86_RESERVED_1 : BYTE ;	//Reserved for system
  OB86_RESERVED_2 : BYTE ;	//Reserved for system
  OB86_MDL_ADDR : WORD ;	//Depending on fault identification code
  OB86_RACKS_FLTD : ARRAY  [0 .. 31 ] OF BOOL ;	//Racks in fault
  OB86_DATE_TIME : DATE_AND_TIME ;	//Date and time OB86 started
END_VAR
BEGIN
NETWORK
TITLE = Fehlermeldung erzeugen
//Fehlermeldung erzeugen
//
//Fehlercode B#16#C1 : Baugruppenträgerausfall
//
//           B#16#C2 : Baugruppenträgerwiederkehr (Baugruppenträgerausfall gehend 
//                     mit Abweichung Soll-/Istausbau)
//
//           B#16#C3 : Dezentrale Peripherie: Ausfall eines DP-Mastersystems
//
//           B#16#C4 : Ausfall einer DP-Station
//
//           B#16#C5 : Störung einer DP-Station
//
      A(;
      L     #OB86_EV_CLASS;
      L     B#16#39;	// kommendes Ereignis
      ==I;
      );
      A(;
      L     #OB86_FLT_ID;
      L     B#16#0;
      <>I;
      );
      =     DB3.DBX 30.6;
      L     #OB86_FLT_ID;
      T     DB3.DBB 40;
END_ORGANIZATION_BLOCK

ORGANIZATION_BLOCK OB 87
TITLE = Kommunikationsfehler
//Erstellung:
//Datum        Bearbeiter                                                 Version
//--------------------------------------------------------------------------------
//03.06.98     Rainer Schaffert (sra)                                     01.00.00
//
//Änderungen:
//Nr. Datum    Bearb Beschreibung                                   Marke Version
//--------------------------------------------------------------------------------
//01  
//
//________________________________________________________________________________
//OB wird bei Kommunikationsfehler bearbeitet
//
AUTHOR : sra
FAMILY : AZO
VERSION : 0.0
VAR_TEMP
  OB87_EV_CLASS : BYTE ;	//16#35 Event class 3
  OB87_FLT_ID : BYTE ;	//16#XX, Fault identifcation code
  OB87_PRIORITY : BYTE ;	//26 (Priority of 1 is lowest)
  OB87_OB_NUMBR : BYTE ;	//87 (Organization block 87, OB87)
  OB87_RESERVED_1 : BYTE ;	//Reserved for system
  OB87_RESERVED_2 : BYTE ;	//Reserved for system
  OB87_RESERVED_3 : WORD ;	//Reserved for system
  OB87_RESERVED_4 : DWORD ;	//Reserved for system
  OB87_DATE_TIME : DATE_AND_TIME ;	//Date and time OB87 started
END_VAR
BEGIN
NETWORK
TITLE = Fehlermeldung erzeugen
//Fehlermeldung erzeugen
//
//Fehlercode B#16#D2 : Senden der Diagnoseeinträge nicht möglich
//
//           B#16#D3 : Synchronisationsdiagramme können nicht gesendet werden
//
//           B#16#D4 : Unzulässiger Uhrzeitsprung durch Uhrzeitsynchronisation
//
//           B#16#D5 : Fehler bei Übernahme der Synchronisationszeit
//
//           B#16#E1 : Falsche Telegrammkennung bei Globaldatenkommunikation
//
//           B#16#E3 : Telegrammlängenfehler bei Globaldatenkommunikation
//
//           B#16#E4 : Unzulässige GD-Paketnummer empfangen
//
//           B#16#E2 : GD-Paketstatus ist nicht in einen DP-eintragbar
//
//           B#16#E5 : Fehler bei Zugriff auf DB beim Datenaustausch über 
//                     Kommunikationsfunktionsbausteine
//
//           B#16#E6 : GD-Gesamtstatus ist nicht in DB eintragbar
//
      L     #OB87_FLT_ID;
      L     B#16#0;
      <>I;
      =     DB3.DBX 30.7;
      L     #OB87_FLT_ID;
      T     DB3.DBB 41;
END_ORGANIZATION_BLOCK

ORGANIZATION_BLOCK OB 100
TITLE = Neustart
//Erstellung:
//Datum        Bearbeiter                                                 Version
//--------------------------------------------------------------------------------
//04.09.2001   R.Schaffert (sra)                                          01.00.00
//  
//Änderungen:
//Nr. Datum    Bearb Änderung                                       Marke  Version
//--------------------------------------------------------------------------------
//01  24.04.17 gea  set service mode lock auto                      (001) 01.00.01
//________________________________________________________________________________
//Programm wird am Anfang von OB 1 fortgesetzt
AUTHOR : sra
FAMILY : AZO
VERSION : 0.0
VAR_TEMP
  OB100_EV_CLASS : BYTE ;	//16#13, Event class 1, Entering event state, Event logged in diagnostic buffer
  OB100_STRTUP : BYTE ;	//16#81/82/83/84 Method of startup
  OB100_PRIORITY : BYTE ;	//27 (Priority of 1 is lowest)
  OB100_OB_NUMBR : BYTE ;	//100 (Organization block 100, OB100)
  OB100_RESERVED_1 : BYTE ;	//Reserved for system
  OB100_RESERVED_2 : BYTE ;	//Reserved for system
  OB100_STOP : WORD ;	//Event that caused CPU to stop (16#4xxx)
  OB100_STRT_INFO : DWORD ;	//Information on how system started
  OB100_DATE_TIME : DATE_AND_TIME ;	//Date and time OB100 started
END_VAR
BEGIN
NETWORK
TITLE = Neustartmerker setzen
      SET;
      S     M 1.3;
      SET;	// (001)
      S     M 9.5;	// (001)
END_ORGANIZATION_BLOCK

ORGANIZATION_BLOCK OB 121
TITLE = Programmierfehler-OB
//Erstellung:
//Datum        Bearbeiter                                                 Version
//--------------------------------------------------------------------------------
//03.06.98     Rainer Schaffert (sra)                                     01.00.00
//
//Änderungen:
//Nr. Datum    Bearb Beschreibung                                   Marke Version
//--------------------------------------------------------------------------------
//01  
//
//________________________________________________________________________________
//OB wird aufgerufen wenn ein Fehler während der Programmbearbeitung auftritt
AUTHOR : sra
FAMILY : AZO
VERSION : 0.0
VAR_TEMP
  OB121_EV_CLASS : BYTE ;	//16#25, Event class 2, Entering event state, Internal fault event
  OB121_SW_FLT : BYTE ;	//16#XX Software programming fault
  OB121_PRIORITY : BYTE ;	//X = Priority of OB where fault occured (Priority of 1 is lowest)
  OB121_OB_NUMBR : BYTE ;	//121 (Organization block 121, OB121)
  OB121_BLK_TYPE : BYTE ;	//16#88/8A/8B/8C/8E Type of block fault occured in
  OB121_RESERVED_1 : BYTE ;	//Reserved for system
  OB121_FLT_REG : WORD ;	//16#XX Specific register that caused fault
  OB121_BLK_NUM : WORD ;	//Number of block that programming fault occured in
  OB121_PRG_ADDR : WORD ;	//Address in block where programming fault occured
  OB121_DATE_TIME : DATE_AND_TIME ;	//Date and time OB121 started
END_VAR
BEGIN
NETWORK
TITLE = Fehlermeldung erzeugen
//Fehlermeldung erzeugen
//
//Fehlercode B#16#21 : BCD-Konvertierungsfehler
//                                
//           B#16#22 : Bereichslängenfehler bei lesen
//
//           B#16#23 : Bereichslängenfehler bei schreiben
//
//           B#16#28 : lesender Zugriff auf ein Byte, Wort oder Doppelwort mit 
//                     einem Pointer, dessen Bitadresse ungleich 0 ist.
//
//           B#16#29 : schreibender Zugriff auf ein Byte, Wort oder Doppelwort 
//                     mit einem Pointer, dessen Bitadresse ungleich 0 ist.
//
//           B#16#24 : Bereichsfehler bei lesen
//
//           B#16#25 : Bereichsfehler bei schreiben
//
//           B#16#26 : Fehler bei Timernummer
//
//           B#16#27 : Fehler bei Zählernummer
//
//           B#16#30 : Schreibender Zugriff auf einen schreibgeschützten Global-DB
//
//           B#16#31 : Schreibender Zugriff auf einen schreibgeschützten 
//                     Instanz-DB
//
//           B#16#32 : DB-Nummernfehler beim Zugriff auf einen Global-DB
//
//           B#16#33 : DB-Nummernfehler beim Zugriff auf einen Instanz-DB
//
//
//
//Fehlermeldung erzeugen
//
//Fehlercode B#16#21 : BCD-Konvertierungsfehler
//                                
//           B#16#22 : Bereichslängenfehler bei lesen
//
//           B#16#23 : Bereichslängenfehler bei schreiben
//
//           B#16#28 : lesender Zugriff auf ein Byte, Wort oder Doppelwort mit 
//                     einem Pointer, dessen Bitadresse ungleich 0 ist.
//
//           B#16#29 : schreibender Zugriff auf ein Byte, Wort oder Doppelwort 
//mit 
//                     einem Pointer, dessen Bitadresse ungleich 0 ist.
//
//           B#16#24 : Bereichsfehler bei lesen
//
//           B#16#25 : Bereichsfehler bei schreiben
//
//           B#16#26 : Fehler bei Timernummer
//
//           B#16#27 : Fehler bei Zählernummer
//
//           B#16#30 : Schreibender Zugriff auf einen schreibgeschützten Global-DB
//
//           B#16#31 : Schreibender Zugriff auf einen schreibgeschützten 
//                     Instanz-DB
//
//           B#16#32 : DB-Nummernfehler beim Zugriff auf einen Global-DB
//
//           B#16#33 : DB-Nummernfehler beim Zugriff auf einen Instanz-DB
//
//           B#16#34 : FC-Nummernfehler beim FC-Aufruf
//
//           B#16#35 : FB-Nummernfehler beim FB-Aufruf
//
//           B#16#3A : Zugriff auf einen nicht geladenen DB
//
//           B#16#3C : Zugriff auf einen nicht geladenen FC
//
//           B#16#3D : Zugriff auf einen nicht geladenen SFC
//
//           B#16#3E : Zugriff auf einen nicht geladenen FB
//
//           B#16#3F : Zugriff auf einen nicht geladenen SFB
//
//
      A(;
      L     #OB121_SW_FLT;
      L     B#16#0;
      <>I;
      );
      =     DB3.DBX 31.0;
      L     #OB121_SW_FLT;
      T     DB3.DBB 42;
END_ORGANIZATION_BLOCK
